{attribute 'no_check'}
// Control Danfoss frequency converter in FC mode
FUNCTION_BLOCK EcFcDS402_DanfossVLT302 EXTENDS EcFcDS402_ComBase IMPLEMENTS I_ActuatorFwdRev
VAR_INPUT
	VeloReference											: 	LREAL := 0.0;  	//[RPM] reference velocity
	RampUp													:	LREAL := 1.0;	//[s] sets slope of ramp
	RampDown												:	LREAL := 1.0;	//[s] sets slope of ramp
 
END_VAR                     							
VAR_OUTPUT                  							
	CiA_Control												:	CiA_DS402Controlword_Danfoss;
	CiA_Status												:	CiA_DS402Statusword_Danfoss;
	ErrorCode										AT  %I*	:	UDINT; 			//1690: see also Danfoss documentation
	OpHours											AT  %I* : 	UDINT;			//1500: Operating Hours
	ActPower												: 	LREAL;			//actual scaled Power of drive 
	ActVelo													: 	LREAL;			//actual scaled velocity of drive
	ActCurrent												: 	LREAL;			//actual current consumption of drive
	Q_TargetVelo									AT  %Q* : 	INT;			//1682: Frequence converter set value velocity
	Q_RampUp										AT  %Q* :	UDINT;			// 341: Frequence converter ramp time up
	Q_RampDown										AT  %Q* :	UDINT;			// 342: Frequence converter ramp time down 
END_VAR                 							
VAR (* IO Internal *)   							
                        							
	_ActVelo										AT  %I* : 	INT; 			//1605: Frequence converter actual velocity in digits based on VeloReference
	_ActCurrent										AT  %I* : 	DINT;			//1614: actual current consumption of drive
	_Power											AT  %I* : 	DINT;			//1610: Power 
END_VAR                 								
VAR                     	
END_VAR

(* Com Danfoss VLT302 over Ethercat Gateway MCA 124 	V1.0	 	*)
// ******************************************************************
{info 'FB EcFcDS402_DanfossVLT302: set parameter 4-10 to [2] both directions'}

(* Protection Switch *******************************************)		
	IF ResetTrig  
	THEN 
		REset(); 
	END_IF
	
	ProtSwitchOK();	
	FuseBrakeOK(); (* same parameter like ProtSwitch *)

(* Contactor ***************************************************)
	Q_Contactor 											:= Contactor AND ProtSwitchOK.Q AND FuseBrakeOK.Q;

(* Read status *************************************************)
	CiA_Status.readStatusword(Statusword);

(* interpret status word ***************************************)
	ActVelo													:= SCALE(_ActVelo, -16384, 16384, -VeloReference, VeloReference);	//16#F000 = -16384 | 16#4000 = 16384    
	ActCurrent             									:= TO_LREAL(_ActCurrent) / 100.0;
	ActPower												:= TO_LREAL(_Power) / 100.0;
	
	Ready													:= CiA_Status.ReadyToSwitchOn AND Q_Contactor;
	Error													:= CiA_Status.Fault AND Q_Contactor;                       									
	Busy													:= CiA_Status.OperationEnabled AND ActVelo <> 0; 
	                                        
// write contorlword DS 402  ****************************************
	CiA_Control.SwitchOn									:= Enable AND Q_Contactor;
	CiA_Control.EnableOperation								:= FeedBwd AND StartBwd AND NOT Start OR Feed AND Start AND NOT StartBwd;
	CiA_Control.FaultReset									:= ResetIntern;
	
	CiA_Control.EnableRamp			 						:= TRUE;
	CiA_Control.RunEnable									:= CiA_Control.SwitchOn;							       
	CiA_Control.Start										:= CiA_Control.EnableOperation;						                     	
	CiA_Control.Reversing			 						:= Start AND NOT StartBwd;	// 15 Reverse     
			
(* setvalue ***************************************************)
	IF CiA_Control.EnableOperation
	THEN
		Q_TargetVelo										:= TO_INT(SCALE(Velo, 	0, VeloReference, 0, 16384));
	ELSE
		Q_TargetVelo										:= 0;
	END_IF
	
	Q_RampUp 												:= TO_UDINT(RampUp*100);
	Q_RampDown 												:= TO_UDINT(RampDown*100);
	              
// Reset FALSE ****************************************************
	ResetIntern												:= FALSE;
	
(* HmiStatus **************************************************)
	Status.0 												:= CiA_Status.OperationEnabled AND StartBwd; 	// counter-clockwise rotation
	Status.1 												:= CiA_Status.OperationEnabled AND Start; 	// clockwise rotation
	Status.2 												:= ActVelo < 0;
	Status.3												:= ActVelo > 0;
	Status.4 												:= FeedBwd;
	Status.5 												:= Feed;
	Status.6 												:= Ready;
	Status.7 												:= Error;
// ****************************************************************

{attribute 'monitoring' := 'call'}
PROPERTY public forwardStarted : BOOL
GET
forwardStarted := CiA_Control.EnableOperation and Q_TargetVelo > 0;
END_GET
END_PROPERTY

{attribute 'monitoring' := 'call'}
PROPERTY public isDisabled : BOOL
GET
isDisabled := not CiA_Status.SwitchedOn and not CiA_Status.OperationEnabled;
END_GET
END_PROPERTY

{attribute 'monitoring' := 'call'}
PROPERTY public isEnabled : BOOL
GET
isEnabled := CiA_Status.SwitchedOn or CiA_Status.OperationEnabled;
END_GET
END_PROPERTY

{attribute 'monitoring' := 'call'}
PROPERTY public isOff : BOOL
GET
isOff := NOT CiA_Status.OperationEnabled;
END_GET
END_PROPERTY

{attribute 'monitoring' := 'call'}
PROPERTY public isOn : BOOL
GET
isOn := CiA_Status.OperationEnabled;
END_GET
END_PROPERTY

{attribute 'monitoring' := 'call'}
PROPERTY public reverseStarted : BOOL
GET
reverseStarted := CiA_Control.EnableOperation and Q_TargetVelo < 0;
END_GET
END_PROPERTY

METHOD setDisable : BOOL
VAR_INPUT
END_VAR

SetDisable													:= Super^.setDisable() AND NOT CiA_Status.SwitchedOn;
END_METHOD

METHOD setEnable : BOOL
VAR_INPUT
END_VAR

SetEnable													:= SUPER^.setEnable() AND CiA_Status.SwitchedOn;
END_METHOD

METHOD PUBLIC startForward : bool //Return busy flag
VAR_INPUT
END_VAR
Start 														:= TRUE; 
StartBwd 													:= FALSE;
startForward												:= Busy and Q_TargetVelo > 0;
END_METHOD

METHOD PUBLIC startReverse : bool //Return busy flag
VAR_INPUT
END_VAR
Start 														:= FALSE; 
StartBwd 													:= TRUE;
startReverse												:= Busy and Q_TargetVelo < 0;
END_METHOD

METHOD PUBLIC switchOn : BOOL  //True if motor is switched on
VAR_INPUT
END_VAR
switchOn := startForward();
END_METHOD

END_FUNCTION_BLOCK

(* stored: Version 1.1.0.1, ProductVersion 3.1.4024.13
   POU EcFcDS402_DanfossVLT302: Id {6a61ff79-e39c-4f94-854b-b9b27ee8042c}, SpecialFunc None
   Folder methods: Id {761efc2e-f347-4cf1-90a1-ffce3ffce262}
   Folder properties: Id {4e300e6c-c6b8-4557-9c20-0d95ede8420a}
   Property forwardStarted: Id {10e691c6-bf76-4fe7-9842-4b57bf71fc38}
   Get Get: Id {8f7cb92b-817e-4f1b-a186-6a75f1492bb2}
   Property isDisabled: Id {72d23790-b63e-4fea-8ce5-78bb38325b54}
   Get Get: Id {001a3371-7acb-4b24-a576-fc2bd325a8ee}
   Property isEnabled: Id {fb874c7c-9a53-49fb-b149-22dfb83b4883}
   Get Get: Id {bdd9d850-af82-490b-aa24-356fd5216ea9}
   Property isOff: Id {62d4f402-a9a2-4830-91b8-30a15217694b}
   Get Get: Id {9f9aa466-f1ec-479c-8b81-10f8b6f3a75b}
   Property isOn: Id {be36e746-fef8-40fa-b4b3-9f89cc48ad98}
   Get Get: Id {a3119b9c-91b5-4855-9b94-5bd311b1e0e0}
   Property reverseStarted: Id {0fe0b9c1-d27a-4872-94ba-5d1ada02be4b}
   Get Get: Id {1c499a9d-f6ea-45cd-aee3-2ba1da2aa4ad}
   Method setDisable: Id {2dbe58eb-2d50-40e4-b60a-db7b7cee9d7a}
   Method setEnable: Id {d9765201-7122-48cc-8faf-b2abfa5d7164}
   Method startForward: Id {6497c166-77b9-42d7-91c7-3a202c067234}
   Method startReverse: Id {232bb19d-4abe-47cd-b73d-758edf012b79}
   Method switchOn: Id {253c23fc-239b-4ca4-b0e8-d1976a61e6e5} *)
